(* CODESYS project mobject-deserialization.library
   Company: mobject
   DefaultNamespace: mobject-deserialization
   Version: 0.1.0
   Placeholder: mobject-deserialization
   Author: mobject dev team
   Title: mobject-deserialization

Project tree, tasks and I/O mapping:
  libraries: mobject-collections, 1.1.0 (mobject); mobject-disposable, 1.0.0 (mobject); mobject-enumerable, 1.1.0 (mobject); mobject-errors, 0.2.0 (mobject); mobject-serialization, 0.4.0 (mobject); Tc2_Standard, * (Beckhoff Automation GmbH); Tc2_System, * (Beckhoff Automation GmbH)
  DeserializationFeedback/
    function block DeserializerFeedback [ST]: FB_exit, DisposeErrors, FirstError, HasError, LogError, Reset, SerializeWith
  Errors/
    IncorrectType/
      function block IncorrectKeyTypeDeserializationError [ST]: FB_init, Message
      function block IncorrectTypeDeserializationError [ST]: FB_init, ErrorType, Message
    Invalid Key/
      function block InvalidKeyDeserializationError [ST]: ErrorType, Message
    Missing Key/
      function block MissingKeyDeserializationError [ST]: FB_init, ErrorType, Message
    function block DeserializationErrorFactory [ST]: CreateIncorrectKeyTypeError, CreateIncorrectTypeError, CreateInvalidKeyError, CreateMissingKeyError
  GarbageCollector/
    function block DeserializerGarbageCollector [ST]: FB_exit, DisposeAll, Deregister, Execute, Register
    interface I_DeserializerGarbageCollector: Deregister, Register
  Interfaces/
    interface I_Deserializable: TryDeserializeFrom
    interface I_Deserializer: Clone, GetArray, GetArrayEnumerator, GetElementByIndex, GetKeyArray, GetKeyObject, GetObject, GetObjectEnumerator, TryDeserializeKeyToObject, TryDeserializeToObject, TryGetBase64, TryGetBool, TryGetByte, TryGetDateTime, TryGetDcTime, TryGetDint, TryGetDword, TryGetFileTime, TryGetHexAsBytes, TryGetInt, TryGetKeyBase64, TryGetKeyBool, TryGetKeyByte, TryGetKeyDateTime, TryGetKeyDcTime, TryGetKeyDint, TryGetKeyDword, TryGetKeyFileTime, TryGetKeyHexAsBytes, TryGetKeyInt, TryGetKeyLint, TryGetKeyLreal, TryGetKeyLtime, TryGetKeyLword, TryGetKeyReal, TryGetKeySint, TryGetKeyString, TryGetKeyTime, TryGetKeyTod, TryGetKeyUdint, TryGetKeyUint, TryGetKeyUlint, TryGetKeyUsint, TryGetKeyWord, TryGetLint, TryGetLreal, TryGetLtime, TryGetLword, TryGetReal, TryGetSint, TryGetString, TryGetTime, TryGetTod, TryGetUdint, TryGetUint, TryGetUlint, TryGetUsint, TryGetWord
    interface I_DeserializerArrayForwardEnumerator: Current, Index, IsValid, MoveNext
    interface I_DeserializerFeedback: LogError
    interface I_DeserializerObjectForwardEnumerator: Current, IsValid, Key, MoveNext
*)

// DeserializationFeedback/DeserializerFeedback
{attribute 'linkalways'} 
{attribute 'no_explicit_call' := 'This FB is a CLASS and must be accessed using methods or properties'}
{attribute 'enable_dynamic_creation'}
FUNCTION_BLOCK DeserializerFeedback IMPLEMENTS I_DeserializerFeedback
VAR
	errors : Stack;
	_hasError : BOOL;
	nullError : NullError;
END_VAR

METHOD FB_exit : BOOL
VAR_INPUT
	bInCopyCode : BOOL; // if TRUE, the exit method is called for exiting an instance that is copied afterwards (online change).
END_VAR
IF bInCopyCode THEN
	RETURN;
END_IF

DisposeErrors();
END_METHOD

METHOD PRIVATE DisposeErrors : BOOL
VAR
	error : I_Error;
END_VAR
WHILE errors.TryPop(error) DO
	error.Dispose();
END_WHILE
END_METHOD

PROPERTY PUBLIC FirstError : I_Error
GET
VAR
	error : I_Error;
END_VAR
IF NOT HasError THEN
	FirstError := nullError;
	RETURN;
END_IF

IF NOT errors.TryPeek(error) THEN
	FirstError := nullError;
	RETURN;
END_IF

FirstError := error;
END_GET
END_PROPERTY

PROPERTY PUBLIC HasError : BOOL
GET
HasError := _hasError;
END_GET
END_PROPERTY

METHOD PUBLIC LogError
VAR_INPUT
	Error : I_Error;
END_VAR
errors.Push(Error);
_hasError := TRUE;
END_METHOD

METHOD PUBLIC Reset : BOOL
VAR_INPUT
END_VAR
DisposeErrors();
_hasError := FALSE;
END_METHOD

METHOD PUBLIC SerializeWith
VAR_INPUT
	Serializer : I_Serializer;
END_VAR
VAR
	enumerator : I_ForwardEnumerator;
	error : I_Error;
END_VAR
IF NOT HasError THEN
	RETURN;
END_IF

Serializer.AddKey('errors');
Serializer.StartArray();

enumerator := errors.GetEnumerator();

WHILE enumerator.MoveNext() DO
	IF enumerator.TryGet(error) THEN
		error.SerializeWith(Serializer);
	END_IF
END_WHILE

enumerator.Dispose();
Serializer.EndArray();
END_METHOD

END_FUNCTION_BLOCK

// Interfaces/I_DeserializerFeedback
INTERFACE I_DeserializerFeedback

METHOD PUBLIC LogError
VAR_INPUT
	Error : I_Error;
END_VAR
END_METHOD

END_INTERFACE

// Errors/IncorrectType/IncorrectKeyTypeDeserializationError
{attribute 'linkalways'} 
{attribute 'no_explicit_call' := 'This FB is a CLASS and must be accessed using methods or properties'}
{attribute 'enable_dynamic_creation'}
FUNCTION_BLOCK IncorrectKeyTypeDeserializationError EXTENDS IncorrectTypeDeserializationError
VAR
	key : T_MAXSTRING;
END_VAR

METHOD FB_init : BOOL
VAR_INPUT
	bInitRetains : BOOL; // if TRUE, the retain variables are initialized (warm start / cold start)
	bInCopyCode : BOOL;  // if TRUE, the instance afterwards gets moved into the copy code (online change)
	DataType : T_MAXSTRING;
	Key : T_MAXSTRING;
END_VAR
THIS^.key := Key;
END_METHOD

PROPERTY PUBLIC Message : T_MAXSTRING
GET
VAR
	messageWithKey : T_MAXSTRING;
END_VAR
messageWithKey := concat(' for key : ',key);
Message := CONCAT(SUPER^.Message, messageWithKey);
END_GET
END_PROPERTY

END_FUNCTION_BLOCK

// Errors/IncorrectType/IncorrectTypeDeserializationError
{attribute 'linkalways'} 
{attribute 'no_explicit_call' := 'This FB is a CLASS and must be accessed using methods or properties'}
{attribute 'enable_dynamic_creation'}
FUNCTION_BLOCK IncorrectTypeDeserializationError EXTENDS Error
VAR
	dataType : T_MAXSTRING;
END_VAR

METHOD FB_init : BOOL
VAR_INPUT
	bInitRetains : BOOL; // if TRUE, the retain variables are initialized (warm start / cold start)
	bInCopyCode : BOOL;  // if TRUE, the instance afterwards gets moved into the copy code (online change)
	DataType : T_MAXSTRING;
END_VAR
THIS^.dataType := DataType;
END_METHOD

PROPERTY PUBLIC ErrorType : T_MAXSTRING
GET
ErrorType := 'INCORRECT_DATATYPE_DESERIALIZATION_ERROR';
END_GET
END_PROPERTY

PROPERTY PUBLIC Message : T_MAXSTRING
GET
Message := CONCAT('Deserialization Failed, Incorrect Datatype : ', dataType);
END_GET
END_PROPERTY

END_FUNCTION_BLOCK

// Errors/Invalid Key/InvalidKeyDeserializationError
{attribute 'linkalways'} 
{attribute 'no_explicit_call' := 'This FB is a CLASS and must be accessed using methods or properties'}
{attribute 'enable_dynamic_creation'}
FUNCTION_BLOCK InvalidKeyDeserializationError EXTENDS Error
VAR
END_VAR

PROPERTY PUBLIC ErrorType : T_MAXSTRING
GET
ErrorType := 'INVALID_KEY_DESERIALIZATION_ERROR';
END_GET
END_PROPERTY

PROPERTY PUBLIC Message : T_MAXSTRING
GET
Message := 'Deserialization Failed, Key Cannot Be Empty';
END_GET
END_PROPERTY

END_FUNCTION_BLOCK

// Errors/Missing Key/MissingKeyDeserializationError
{attribute 'linkalways'} 
{attribute 'no_explicit_call' := 'This FB is a CLASS and must be accessed using methods or properties'}
{attribute 'enable_dynamic_creation'}
FUNCTION_BLOCK MissingKeyDeserializationError EXTENDS Error
VAR
	key : T_MAXSTRING;
END_VAR

METHOD FB_init : BOOL
VAR_INPUT
	bInitRetains : BOOL; // if TRUE, the retain variables are initialized (warm start / cold start)
	bInCopyCode : BOOL;  // if TRUE, the instance afterwards gets moved into the copy code (online change)
	Key : T_MAXSTRING;
END_VAR
this^.key := Key;
END_METHOD

PROPERTY PUBLIC ErrorType : T_MAXSTRING
GET
ErrorType := 'MISSING_KEY_DESERIALIZATION_ERROR';
END_GET
END_PROPERTY

PROPERTY PUBLIC Message : T_MAXSTRING
GET
Message := CONCAT('Deserialization Failed, Missing Key : ',key);
END_GET
END_PROPERTY

END_FUNCTION_BLOCK

// Errors/DeserializationErrorFactory
{attribute 'linkalways'} 
{attribute 'no_explicit_call' := 'This FB is a CLASS and must be accessed using methods or properties'}
{attribute 'enable_dynamic_creation'}
FUNCTION_BLOCK DeserializationErrorFactory
VAR
END_VAR

METHOD PUBLIC CreateIncorrectKeyTypeError : I_Error
VAR_INPUT
	ExpectedType : T_MAXSTRING;
	ActualKey : T_MAXSTRING;
END_VAR
VAR
	pError : POINTER TO IncorrectKeyTypeDeserializationError;
END_VAR
pError := __NEW(IncorrectKeyTypeDeserializationError(DataType := ExpectedType, Key := ActualKey));
CreateIncorrectKeyTypeError := pError^;
END_METHOD

METHOD PUBLIC CreateIncorrectTypeError : I_Error
VAR_INPUT
	ExpectedType : T_MAXSTRING;
END_VAR
VAR
	pError : POINTER TO IncorrectTypeDeserializationError;
END_VAR
pError := __NEW(IncorrectTypeDeserializationError(DataType := ExpectedType));
CreateIncorrectTypeError := pError^;
END_METHOD

METHOD PUBLIC CreateInvalidKeyError : I_Error
VAR_INPUT
END_VAR
VAR
	pError : POINTER TO InvalidKeyDeserializationError;
END_VAR
pError := __NEW(InvalidKeyDeserializationError);
CreateInvalidKeyError := pError^;
END_METHOD

METHOD PUBLIC CreateMissingKeyError : I_Error
VAR_INPUT
	ExpectedKey : T_MAXSTRING;
END_VAR
VAR
	pError : POINTER TO MissingKeyDeserializationError;
END_VAR
pError := __NEW(MissingKeyDeserializationError(Key := ExpectedKey));
CreateMissingKeyError := pError^;
END_METHOD

END_FUNCTION_BLOCK

// GarbageCollector/DeserializerGarbageCollector
{attribute 'linkalways'} 
{attribute 'no_explicit_call' := 'This FB is a CLASS and must be accessed using methods or properties'}
{attribute 'enable_dynamic_creation'}
FUNCTION_BLOCK DeserializerGarbageCollector EXTENDS Disposable Implements I_DeserializerGarbageCollector
VAR
	deserializers : Stack;
END_VAR

METHOD FB_exit : BOOL
VAR_INPUT
	bInCopyCode : BOOL; // if TRUE, the exit method is called for exiting an instance that is copied afterwards (online change).
END_VAR
IF bInCopyCode THEN
	RETURN;
END_IF

DisposeAll();
END_METHOD

METHOD PROTECTED DisposeAll
VAR
	deserializer : I_Deserializer;
END_VAR
WHILE deserializers.TryPop(deserializer) DO
	deserializer.Dispose();
END_WHILE
END_METHOD

METHOD PUBLIC Deregister
VAR_INPUT
	Deserializer : I_Deserializer;
END_VAR
deserializers.TryRemoveItem(Deserializer);
END_METHOD

METHOD PUBLIC Execute
VAR_INPUT
END_VAR
DisposeAll();
END_METHOD

METHOD PUBLIC Register
VAR_INPUT
	Deserializer : I_Deserializer;
END_VAR
deserializers.Push(Deserializer);
END_METHOD

END_FUNCTION_BLOCK

// GarbageCollector/I_DeserializerGarbageCollector
INTERFACE I_DeserializerGarbageCollector EXTENDS __SYSTEM.IQueryInterface

METHOD PUBLIC Deregister
VAR_INPUT
	Deserializer : I_Deserializer;
END_VAR
END_METHOD

METHOD PUBLIC Register
VAR_INPUT
	Deserializer : I_Deserializer;
END_VAR
END_METHOD

END_INTERFACE

// Interfaces/I_Deserializer
INTERFACE I_Deserializer EXTENDS I_Disposable

METHOD PUBLIC Clone : I_Deserializer
END_METHOD

METHOD GetArray : I_Deserializer
VAR_INPUT
END_VAR
END_METHOD

METHOD GetArrayEnumerator : I_DeserializerArrayForwardEnumerator
VAR_INPUT
END_VAR
END_METHOD

METHOD GetElementByIndex : I_Deserializer
VAR_INPUT
	Index : UDINT;
END_VAR
END_METHOD

METHOD GetKeyArray : I_Deserializer
VAR_INPUT
	Key : T_MAXSTRING;
END_VAR
END_METHOD

METHOD GetKeyObject : I_Deserializer
VAR_INPUT
	Key : T_MAXSTRING;
END_VAR
END_METHOD

METHOD GetObject : I_Deserializer
VAR_INPUT
END_VAR
END_METHOD

METHOD GetObjectEnumerator : I_DeserializerObjectForwardEnumerator
VAR_INPUT
END_VAR
END_METHOD

METHOD TryDeserializeKeyToObject : BOOL
VAR_INPUT
	Key : T_MAXSTRING;
	Object : I_Deserializable;
	Feedback : I_DeserializerFeedback;
END_VAR
END_METHOD

METHOD TryDeserializeToObject : BOOL
VAR_INPUT
	Object : I_Deserializable;
	Feedback : I_DeserializerFeedback;
END_VAR
END_METHOD

METHOD TryGetBase64 : BOOL
VAR_INPUT
	pBytes : POINTER TO BYTE;
	nBytes : DINT;
	Feedback : I_DeserializerFeedback;
END_VAR
END_METHOD

METHOD TryGetBool : BOOL
VAR_INPUT
	Destination : REFERENCE TO BOOL;
	Feedback : I_DeserializerFeedback;
END_VAR
END_METHOD

METHOD TryGetByte : BOOL
VAR_INPUT
	Destination : REFERENCE TO BYTE;
	Feedback : I_DeserializerFeedback;
END_VAR
END_METHOD

METHOD TryGetDateTime : BOOL
VAR_INPUT
	Destination : REFERENCE TO DATE_AND_TIME;
	Feedback : I_DeserializerFeedback;
END_VAR
END_METHOD

METHOD TryGetDcTime : BOOL
VAR_INPUT
	Destination : REFERENCE TO DCTIME;
	Feedback : I_DeserializerFeedback;
END_VAR
END_METHOD

METHOD TryGetDint : BOOL
VAR_INPUT
	Destination : REFERENCE TO DINT;
	Feedback : I_DeserializerFeedback;
END_VAR
END_METHOD

METHOD TryGetDword : BOOL
VAR_INPUT
	Destination : REFERENCE TO DWORD;
	Feedback : I_DeserializerFeedback;
END_VAR
END_METHOD

METHOD TryGetFileTime : BOOL
VAR_INPUT
	Destination : REFERENCE TO FILETIME;
	Feedback : I_DeserializerFeedback;
END_VAR
END_METHOD

METHOD TryGetHexAsBytes : BOOL
VAR_INPUT
	pBytes : POINTER TO BYTE;
	nBytes : DINT;
	Feedback : I_DeserializerFeedback;
END_VAR
END_METHOD

METHOD TryGetInt : BOOL
VAR_INPUT
	Destination : REFERENCE TO INT;
	Feedback : I_DeserializerFeedback;
END_VAR
END_METHOD

METHOD TryGetKeyBase64 : BOOL
VAR_INPUT
	Key : T_MAXSTRING;
	pBytes : POINTER TO BYTE;
	nBytes : DINT;
	Feedback : I_DeserializerFeedback;
END_VAR
END_METHOD

METHOD TryGetKeyBool : BOOL
VAR_INPUT
	Key : T_MAXSTRING;
	Destination : REFERENCE TO BOOL;
	Feedback : I_DeserializerFeedback;
END_VAR
END_METHOD

METHOD TryGetKeyByte : BOOL
VAR_INPUT
	Key : T_MAXSTRING;
	Destination : REFERENCE TO BYTE;
	Feedback : I_DeserializerFeedback;
END_VAR
END_METHOD

METHOD TryGetKeyDateTime : BOOL
VAR_INPUT
	Key : T_MAXSTRING;
	Destination : REFERENCE TO DATE_AND_TIME;
	Feedback : I_DeserializerFeedback;
END_VAR
END_METHOD

METHOD TryGetKeyDcTime : BOOL
VAR_INPUT
	Key : T_MAXSTRING;
	Destination : REFERENCE TO DCTIME;
	Feedback : I_DeserializerFeedback;
END_VAR
END_METHOD

METHOD TryGetKeyDint : BOOL
VAR_INPUT
	Key : T_MAXSTRING;
	Destination : REFERENCE TO DINT;
	Feedback : I_DeserializerFeedback;
END_VAR
END_METHOD

METHOD TryGetKeyDword : BOOL
VAR_INPUT
	Key : T_MAXSTRING;
	Destination : REFERENCE TO DWORD;
	Feedback : I_DeserializerFeedback;
END_VAR
END_METHOD

METHOD TryGetKeyFileTime : BOOL
VAR_INPUT
	Key : T_MAXSTRING;
	Destination : REFERENCE TO FILETIME;
	Feedback : I_DeserializerFeedback;
END_VAR
END_METHOD

METHOD TryGetKeyHexAsBytes : BOOL
VAR_INPUT
	Key : T_MAXSTRING;
	pBytes : POINTER TO BYTE;
	nBytes : DINT;
	Feedback : I_DeserializerFeedback;
END_VAR
END_METHOD

METHOD TryGetKeyInt : BOOL
VAR_INPUT
	Key : T_MAXSTRING;
	Destination : REFERENCE TO INT;
	Feedback : I_DeserializerFeedback;
END_VAR
END_METHOD

METHOD TryGetKeyLint : BOOL
VAR_INPUT
	Key : T_MAXSTRING;
	Destination : REFERENCE TO LINT;
	Feedback : I_DeserializerFeedback;
END_VAR
END_METHOD

METHOD TryGetKeyLreal : BOOL
VAR_INPUT
	Key : T_MAXSTRING;
	Destination : REFERENCE TO LREAL;
	Feedback : I_DeserializerFeedback;
END_VAR
END_METHOD

METHOD TryGetKeyLtime : BOOL
VAR_INPUT
	Key : T_MAXSTRING;
	Destination : REFERENCE TO LTIME;
	Feedback : I_DeserializerFeedback;
END_VAR
END_METHOD

METHOD TryGetKeyLword : BOOL
VAR_INPUT
	Key : T_MAXSTRING;
	Destination : REFERENCE TO LWORD;
	Feedback : I_DeserializerFeedback;
END_VAR
END_METHOD

METHOD TryGetKeyReal : BOOL
VAR_INPUT
	Key : T_MAXSTRING;
	Destination : REFERENCE TO REAL;
	Feedback : I_DeserializerFeedback;
END_VAR
END_METHOD

METHOD TryGetKeySint : BOOL
VAR_INPUT
	Key : T_MAXSTRING;
	Destination : REFERENCE TO SINT;
	Feedback : I_DeserializerFeedback;
END_VAR
END_METHOD

METHOD TryGetKeyString : BOOL
VAR_INPUT
	Key : T_MAXSTRING;
	Destination : REFERENCE TO STRING;
	Feedback : I_DeserializerFeedback;
END_VAR
END_METHOD

METHOD TryGetKeyTime : BOOL
VAR_INPUT
	Key : T_MAXSTRING;
	Destination : REFERENCE TO TIME;
	Feedback : I_DeserializerFeedback;
END_VAR
END_METHOD

METHOD TryGetKeyTod : BOOL
VAR_INPUT
	Key : T_MAXSTRING;
	Destination : REFERENCE TO TOD;
	Feedback : I_DeserializerFeedback;
END_VAR
END_METHOD

METHOD TryGetKeyUdint : BOOL
VAR_INPUT
	Key : T_MAXSTRING;
	Destination : REFERENCE TO UDINT;
	Feedback : I_DeserializerFeedback;
END_VAR
END_METHOD

METHOD TryGetKeyUint : BOOL
VAR_INPUT
	Key : T_MAXSTRING;
	Destination : REFERENCE TO UINT;
	Feedback : I_DeserializerFeedback;
END_VAR
END_METHOD

METHOD TryGetKeyUlint : BOOL
VAR_INPUT
	Key : T_MAXSTRING;
	Destination : REFERENCE TO ULINT;
	Feedback : I_DeserializerFeedback;
END_VAR
END_METHOD

METHOD TryGetKeyUsint : BOOL
VAR_INPUT
	Key : T_MAXSTRING;
	Destination : REFERENCE TO USINT;
	Feedback : I_DeserializerFeedback;
END_VAR
END_METHOD

METHOD TryGetKeyWord : BOOL
VAR_INPUT
	Key : T_MAXSTRING;
	Destination : REFERENCE TO WORD;
	Feedback : I_DeserializerFeedback;
END_VAR
END_METHOD

METHOD TryGetLint : BOOL
VAR_INPUT
	Destination : REFERENCE TO LINT;
	Feedback : I_DeserializerFeedback;
END_VAR
END_METHOD

METHOD TryGetLreal : BOOL
VAR_INPUT
	Destination : REFERENCE TO LREAL;
	Feedback : I_DeserializerFeedback;
END_VAR
END_METHOD

METHOD TryGetLtime : BOOL
VAR_INPUT
	Destination : REFERENCE TO LTIME;
	Feedback : I_DeserializerFeedback;
END_VAR
END_METHOD

METHOD TryGetLword : BOOL
VAR_INPUT
	Destination : REFERENCE TO LWORD;
	Feedback : I_DeserializerFeedback;
END_VAR
END_METHOD

METHOD TryGetReal : BOOL
VAR_INPUT
	Destination : REFERENCE TO REAL;
	Feedback : I_DeserializerFeedback;
END_VAR
END_METHOD

METHOD TryGetSint : BOOL
VAR_INPUT
	Destination : REFERENCE TO SINT;
	Feedback : I_DeserializerFeedback;
END_VAR
END_METHOD

METHOD TryGetString : BOOL
VAR_INPUT
	Destination : REFERENCE TO STRING;
	Feedback : I_DeserializerFeedback;
END_VAR
END_METHOD

METHOD TryGetTime : BOOL
VAR_INPUT
	Destination : REFERENCE TO TIME;
	Feedback : I_DeserializerFeedback;
END_VAR
END_METHOD

METHOD TryGetTod : BOOL
VAR_INPUT
	Destination : REFERENCE TO TOD;
	Feedback : I_DeserializerFeedback;
END_VAR
END_METHOD

METHOD TryGetUdint : BOOL
VAR_INPUT
	Destination : REFERENCE TO UDINT;
	Feedback : I_DeserializerFeedback;
END_VAR
END_METHOD

METHOD TryGetUint : BOOL
VAR_INPUT
	Destination : REFERENCE TO UINT;
	Feedback : I_DeserializerFeedback;
END_VAR
END_METHOD

METHOD TryGetUlint : BOOL
VAR_INPUT
	Destination : REFERENCE TO ULINT;
	Feedback : I_DeserializerFeedback;
END_VAR
END_METHOD

METHOD TryGetUsint : BOOL
VAR_INPUT
	Destination : REFERENCE TO USINT;
	Feedback : I_DeserializerFeedback;
END_VAR
END_METHOD

METHOD TryGetWord : BOOL
VAR_INPUT
	Destination : REFERENCE TO WORD;
	Feedback : I_DeserializerFeedback;
END_VAR
END_METHOD

END_INTERFACE

// Interfaces/I_DeserializerArrayForwardEnumerator
INTERFACE I_DeserializerArrayForwardEnumerator EXTENDS I_Disposable

PROPERTY PUBLIC Current : I_Deserializer
GET
END_GET
END_PROPERTY

PROPERTY Index : DINT
GET
END_GET
END_PROPERTY

PROPERTY IsValid : BOOL
GET
END_GET
END_PROPERTY

METHOD MoveNext : BOOL
VAR_INPUT
END_VAR
END_METHOD

END_INTERFACE

// Interfaces/I_DeserializerObjectForwardEnumerator
INTERFACE I_DeserializerObjectForwardEnumerator EXTENDS I_Disposable

PROPERTY PUBLIC Current : I_Deserializer
GET
END_GET
END_PROPERTY

PROPERTY IsValid : BOOL
GET
END_GET
END_PROPERTY

PROPERTY Key : T_MAXSTRING
GET
END_GET
END_PROPERTY

METHOD MoveNext : BOOL
VAR_INPUT
END_VAR
END_METHOD

END_INTERFACE

// Interfaces/I_Deserializable
INTERFACE I_Deserializable EXTENDS __SYSTEM.IQueryInterface

METHOD TryDeserializeFrom : BOOL
VAR_INPUT
	Deserializer : I_Deserializer;
	Feedback : I_DeserializerFeedback;
END_VAR
END_METHOD

END_INTERFACE
